// TIA Portal V20 export
FUNCTION "CallAlarmCountMapping" : Void   // FC6, LAD
// stored: SetENOAutomatically false
BEGIN

REGION Network 1: Cutter Life Count
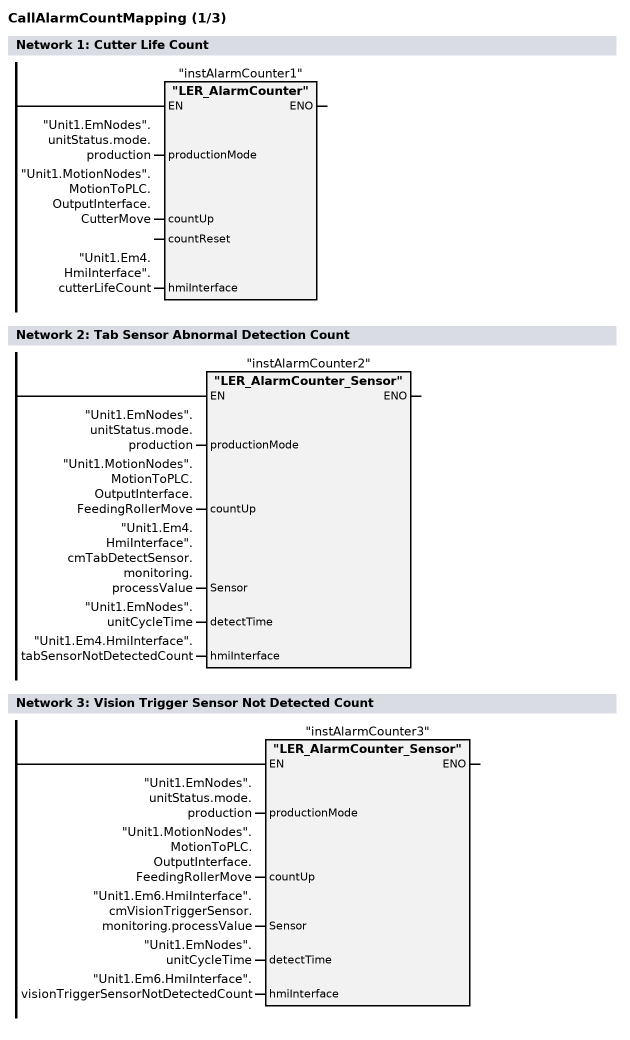
   RUNG wire#powerrail
      "instAlarmCounter1"(productionMode := "Unit1.EmNodes".unitStatus.mode.production, countUp := "Unit1.MotionNodes".MotionToPLC.OutputInterface.CutterMove, countReset :=, hmiInterface := "Unit1.Em4.HmiInterface".cutterLifeCount)
   END_RUNG
   // the same network as SCL:
   "instAlarmCounter1"(productionMode := "Unit1.EmNodes".unitStatus.mode.production,   // "LER_AlarmCounter"
                       countUp := "Unit1.MotionNodes".MotionToPLC.OutputInterface.CutterMove,
                       hmiInterface := "Unit1.Em4.HmiInterface".cutterLifeCount);
END_REGION

REGION Network 2: Tab Sensor Abnormal Detection Count
   RUNG wire#powerrail
      "instAlarmCounter2"(productionMode := "Unit1.EmNodes".unitStatus.mode.production, countUp := "Unit1.MotionNodes".MotionToPLC.OutputInterface.FeedingRollerMove, Sensor := "Unit1.Em4.HmiInterface".cmTabDetectSensor.monitoring.processValue, detectTime := "Unit1.EmNodes".unitCycleTime, hmiInterface := "Unit1.Em4.HmiInterface".tabSensorNotDetectedCount)
   END_RUNG
   // the same network as SCL:
   "instAlarmCounter2"(productionMode := "Unit1.EmNodes".unitStatus.mode.production,   // "LER_AlarmCounter_Sensor"
                       countUp := "Unit1.MotionNodes".MotionToPLC.OutputInterface.FeedingRollerMove,
                       Sensor := "Unit1.Em4.HmiInterface".cmTabDetectSensor.monitoring.processValue,
                       detectTime := "Unit1.EmNodes".unitCycleTime,
                       hmiInterface := "Unit1.Em4.HmiInterface".tabSensorNotDetectedCount);
END_REGION

REGION Network 3: Vision Trigger Sensor Not Detected Count
   RUNG wire#powerrail
      "instAlarmCounter3"(productionMode := "Unit1.EmNodes".unitStatus.mode.production, countUp := "Unit1.MotionNodes".MotionToPLC.OutputInterface.FeedingRollerMove, Sensor := "Unit1.Em6.HmiInterface".cmVisionTriggerSensor.monitoring.processValue, detectTime := "Unit1.EmNodes".unitCycleTime, hmiInterface := "Unit1.Em6.HmiInterface".visionTriggerSensorNotDetectedCount)
   END_RUNG
   // the same network as SCL:
   "instAlarmCounter3"(productionMode := "Unit1.EmNodes".unitStatus.mode.production,   // "LER_AlarmCounter_Sensor"
                       countUp := "Unit1.MotionNodes".MotionToPLC.OutputInterface.FeedingRollerMove,
                       Sensor := "Unit1.Em6.HmiInterface".cmVisionTriggerSensor.monitoring.processValue,
                       detectTime := "Unit1.EmNodes".unitCycleTime,
                       hmiInterface := "Unit1.Em6.HmiInterface".visionTriggerSensorNotDetectedCount);
END_REGION

REGION Network 4: Ng Kicker Sensor Not Detected Count
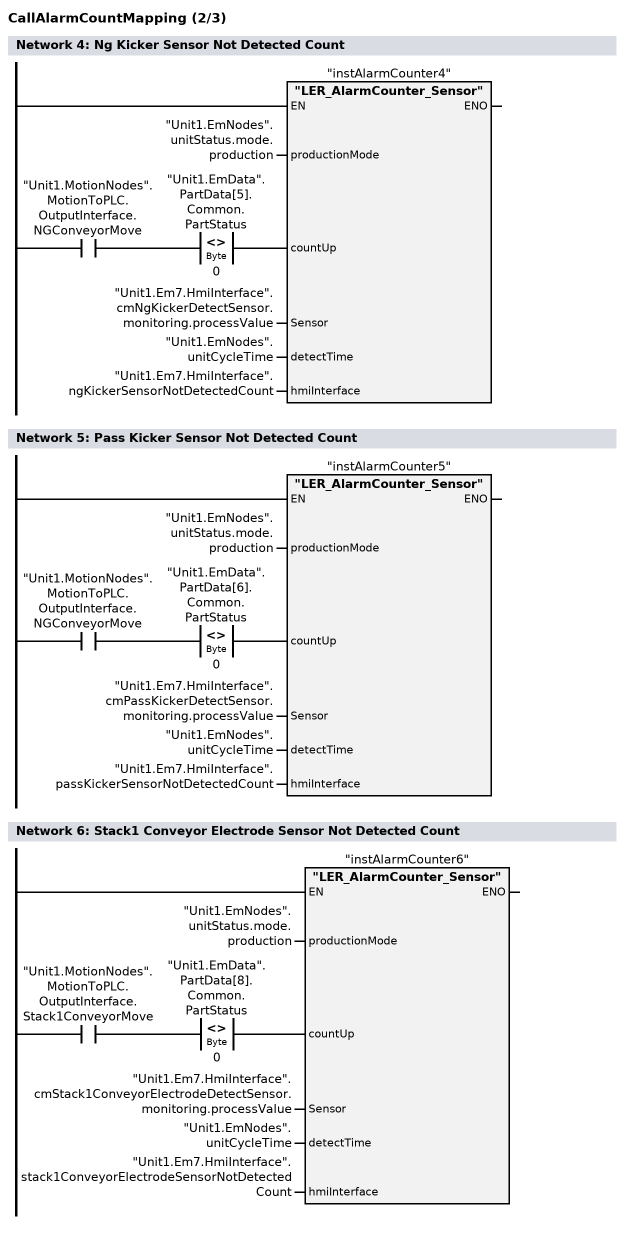
   RUNG wire#powerrail
      "instAlarmCounter4"(countUp := wire#w1, productionMode := "Unit1.EmNodes".unitStatus.mode.production, Sensor := "Unit1.Em7.HmiInterface".cmNgKickerDetectSensor.monitoring.processValue, detectTime := "Unit1.EmNodes".unitCycleTime, hmiInterface := "Unit1.Em7.HmiInterface".ngKickerSensorNotDetectedCount)
   END_RUNG
   RUNG wire#powerrail
      Contact( "Unit1.MotionNodes".MotionToPLC.OutputInterface.NGConveyorMove )
      { S7_Templates := "SrcType := Byte" } NE_Contact(in1 := "Unit1.EmData".PartData[5].Common.PartStatus, in2 := 0)
   END_RUNG wire#w1
   // the same network as SCL:
   "instAlarmCounter4"(productionMode := "Unit1.EmNodes".unitStatus.mode.production,   // "LER_AlarmCounter_Sensor"
                       countUp := "Unit1.MotionNodes".MotionToPLC.OutputInterface.NGConveyorMove AND ("Unit1.EmData".PartData[5].Common.PartStatus <> 0),
                       Sensor := "Unit1.Em7.HmiInterface".cmNgKickerDetectSensor.monitoring.processValue,
                       detectTime := "Unit1.EmNodes".unitCycleTime,
                       hmiInterface := "Unit1.Em7.HmiInterface".ngKickerSensorNotDetectedCount);
END_REGION

REGION Network 5: Pass Kicker Sensor Not Detected Count
   RUNG wire#powerrail
      "instAlarmCounter5"(countUp := wire#w1, productionMode := "Unit1.EmNodes".unitStatus.mode.production, Sensor := "Unit1.Em7.HmiInterface".cmPassKickerDetectSensor.monitoring.processValue, detectTime := "Unit1.EmNodes".unitCycleTime, hmiInterface := "Unit1.Em7.HmiInterface".passKickerSensorNotDetectedCount)
   END_RUNG
   RUNG wire#powerrail
      Contact( "Unit1.MotionNodes".MotionToPLC.OutputInterface.NGConveyorMove )
      { S7_Templates := "SrcType := Byte" } NE_Contact(in1 := "Unit1.EmData".PartData[6].Common.PartStatus, in2 := 0)
   END_RUNG wire#w1
   // the same network as SCL:
   "instAlarmCounter5"(productionMode := "Unit1.EmNodes".unitStatus.mode.production,   // "LER_AlarmCounter_Sensor"
                       countUp := "Unit1.MotionNodes".MotionToPLC.OutputInterface.NGConveyorMove AND ("Unit1.EmData".PartData[6].Common.PartStatus <> 0),
                       Sensor := "Unit1.Em7.HmiInterface".cmPassKickerDetectSensor.monitoring.processValue,
                       detectTime := "Unit1.EmNodes".unitCycleTime,
                       hmiInterface := "Unit1.Em7.HmiInterface".passKickerSensorNotDetectedCount);
END_REGION

REGION Network 6: Stack1 Conveyor Electrode Sensor Not Detected Count
   RUNG wire#powerrail
      "instAlarmCounter6"(countUp := wire#w1, productionMode := "Unit1.EmNodes".unitStatus.mode.production, Sensor := "Unit1.Em7.HmiInterface".cmStack1ConveyorElectrodeDetectSensor.monitoring.processValue, detectTime := "Unit1.EmNodes".unitCycleTime, hmiInterface := "Unit1.Em7.HmiInterface".stack1ConveyorElectrodeSensorNotDetectedCount)
   END_RUNG
   RUNG wire#powerrail
      Contact( "Unit1.MotionNodes".MotionToPLC.OutputInterface.Stack1ConveyorMove )
      { S7_Templates := "SrcType := Byte" } NE_Contact(in1 := "Unit1.EmData".PartData[8].Common.PartStatus, in2 := 0)
   END_RUNG wire#w1
   // the same network as SCL:
   "instAlarmCounter6"(productionMode := "Unit1.EmNodes".unitStatus.mode.production,   // "LER_AlarmCounter_Sensor"
                       countUp := "Unit1.MotionNodes".MotionToPLC.OutputInterface.Stack1ConveyorMove AND ("Unit1.EmData".PartData[8].Common.PartStatus <> 0),
                       Sensor := "Unit1.Em7.HmiInterface".cmStack1ConveyorElectrodeDetectSensor.monitoring.processValue,
                       detectTime := "Unit1.EmNodes".unitCycleTime,
                       hmiInterface := "Unit1.Em7.HmiInterface".stack1ConveyorElectrodeSensorNotDetectedCount);
END_REGION

REGION Network 7: Stack2 Conveyor Electrode Sensor Not Detected Count
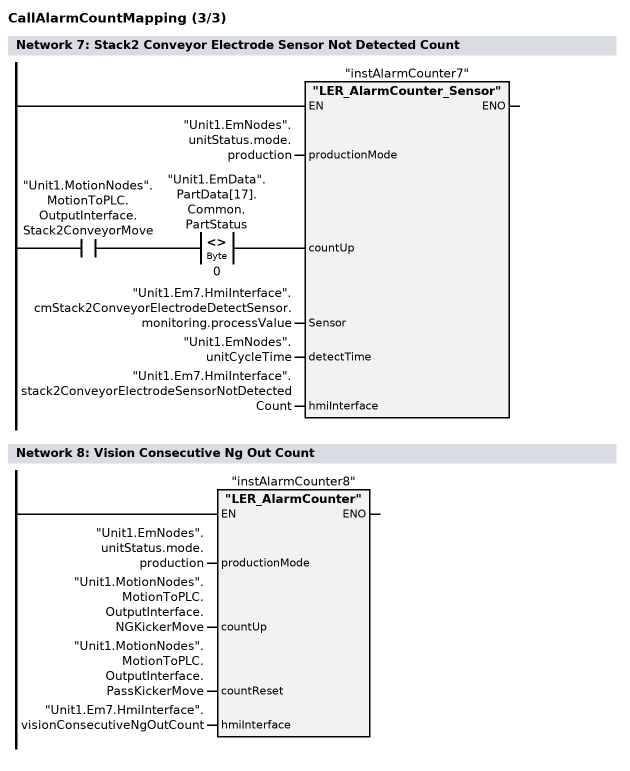
   RUNG wire#powerrail
      "instAlarmCounter7"(countUp := wire#w1, productionMode := "Unit1.EmNodes".unitStatus.mode.production, Sensor := "Unit1.Em7.HmiInterface".cmStack2ConveyorElectrodeDetectSensor.monitoring.processValue, detectTime := "Unit1.EmNodes".unitCycleTime, hmiInterface := "Unit1.Em7.HmiInterface".stack2ConveyorElectrodeSensorNotDetectedCount)
   END_RUNG
   RUNG wire#powerrail
      Contact( "Unit1.MotionNodes".MotionToPLC.OutputInterface.Stack2ConveyorMove )
      { S7_Templates := "SrcType := Byte" } NE_Contact(in1 := "Unit1.EmData".PartData[17].Common.PartStatus, in2 := 0)
   END_RUNG wire#w1
   // the same network as SCL:
   "instAlarmCounter7"(productionMode := "Unit1.EmNodes".unitStatus.mode.production,   // "LER_AlarmCounter_Sensor"
                       countUp := "Unit1.MotionNodes".MotionToPLC.OutputInterface.Stack2ConveyorMove AND ("Unit1.EmData".PartData[17].Common.PartStatus <> 0),
                       Sensor := "Unit1.Em7.HmiInterface".cmStack2ConveyorElectrodeDetectSensor.monitoring.processValue,
                       detectTime := "Unit1.EmNodes".unitCycleTime,
                       hmiInterface := "Unit1.Em7.HmiInterface".stack2ConveyorElectrodeSensorNotDetectedCount);
END_REGION

REGION Network 8: Vision Consecutive Ng Out Count
   RUNG wire#powerrail
      "instAlarmCounter8"(productionMode := "Unit1.EmNodes".unitStatus.mode.production, countUp := "Unit1.MotionNodes".MotionToPLC.OutputInterface.NGKickerMove, countReset := "Unit1.MotionNodes".MotionToPLC.OutputInterface.PassKickerMove, hmiInterface := "Unit1.Em7.HmiInterface".visionConsecutiveNgOutCount)
   END_RUNG
   // the same network as SCL:
   "instAlarmCounter8"(productionMode := "Unit1.EmNodes".unitStatus.mode.production,   // "LER_AlarmCounter"
                       countUp := "Unit1.MotionNodes".MotionToPLC.OutputInterface.NGKickerMove,
                       countReset := "Unit1.MotionNodes".MotionToPLC.OutputInterface.PassKickerMove,
                       hmiInterface := "Unit1.Em7.HmiInterface".visionConsecutiveNgOutCount);
END_REGION
END_FUNCTION
